{attribute 'GeneratedUsingTerminal: EL6201-0000-0017'}
{attribute addProperty BoxType "EL6201-0000-0017"}
{attribute addProperty Id "Slave_8A_DO0BOOL1Slave_8A_DO1BOOL1Slave_8A_DO2BOOL1Slave_8A_DO3BOOL1Slave_8B_DO0BOOL1Slave_8B_DO1BOOL1Slave_8B_DO2BOOL1Slave_8B_DO3BOOL1"}
{attribute addProperty CRC "2246474998"}
{attribute addProperty Size "8"}
TYPE Slave_8_Outputs_85E67CF6 :
STRUCT
	{attribute addProperty Name "Slave_8A_DO0"}
	Slave_8A_DO0 : BOOL;
	{attribute addProperty Name "Slave_8A_DO1"}
	Slave_8A_DO1 : BOOL;
	{attribute addProperty Name "Slave_8A_DO2"}
	Slave_8A_DO2 : BOOL;
	{attribute addProperty Name "Slave_8A_DO3"}
	Slave_8A_DO3 : BOOL;
	{attribute addProperty Name "Slave_8B_DO0"}
	Slave_8B_DO0 : BOOL;
	{attribute addProperty Name "Slave_8B_DO1"}
	Slave_8B_DO1 : BOOL;
	{attribute addProperty Name "Slave_8B_DO2"}
	Slave_8B_DO2 : BOOL;
	{attribute addProperty Name "Slave_8B_DO3"}
	Slave_8B_DO3 : BOOL;
END_STRUCT
END_TYPE

(* stored: Version 1.2.0.0, ProductVersion 3.1.4024.9
   DUT Slave_8_Outputs_85E67CF6: Id {aff1889b-057f-4d85-9c2d-d702f240a3cf} *)
